INTERFACE ITF_BaseLoggerElement EXTENDS ITF_Base

(*			
	EVERDE sp. z o.o.
	Rafał Osajda		24.03.2025		TC 4024.66
	Definicja nowego zgłoszenia
*)
METHOD PUBLIC EventsDefinition : BOOL
END_METHOD

METHOD PUBLIC GetCode : STRING
VAR_INPUT
END_VAR
END_METHOD

METHOD PUBLIC GetID : UINT
VAR_INPUT
END_VAR
END_METHOD

METHOD PUBLIC GetIdentyfier : ST_BaseElementIdentifier
VAR_INPUT
END_VAR
END_METHOD

METHOD PUBLIC GetName : ST_BaseLabel
VAR_INPUT
END_VAR
END_METHOD

METHOD PUBLIC GetType : E_BaseElementType
VAR_INPUT
END_VAR
END_METHOD

METHOD PUBLIC SetCode
VAR_INPUT
	sCode							: STRING;
	sAdd							: STRING;
END_VAR
END_METHOD

(*			
	EVERDE sp. z o.o.
	Rafał Osajda		03.10.2025		TC 4024.66
	nadawanie unikalnych ID dla zdarzeń
*)
METHOD PUBLIC SetEventsIDs : UINT
VAR_INPUT
	uiNewID		: UINT;
END_VAR
END_METHOD

METHOD PUBLIC SetID : UINT
VAR_INPUT
	uiID					: UINT;
END_VAR
END_METHOD

METHOD PUBLIC SetName
VAR_INPUT
	stName				: ST_BaseLabel;
END_VAR
END_METHOD

METHOD PUBLIC SetType
VAR_INPUT
	eType					: E_BaseElementType;
END_VAR
END_METHOD

END_INTERFACE

(* stored: Version 1.1.0.1
   Itf ITF_BaseLoggerElement: Id {040130d5-be8c-0d8f-3758-2f1440aef3cb}
   Folder ID: Id {ebebc54b-7071-0c25-1f06-3769663c0ef5}
   Method EventsDefinition: Id {9fbb4552-8362-0324-08b0-1fb2884dba78}
   Method GetCode: Id {8b6863d7-2a35-07f8-278a-c5063af13d5f}
   Method GetID: Id {01682019-6db3-0ac2-2322-ec1c5cb9c3b3}
   Method GetIdentyfier: Id {9e739503-7893-0bf4-399c-b179c7bd0bc7}
   Method GetName: Id {878e4ebd-33ce-0ec5-047c-9c76b95779fa}
   Method GetType: Id {c399515a-c57b-0d5c-3183-92e3bee5c2f8}
   Method SetCode: Id {709cb346-bc66-0698-2a3d-3e8bbcb515cf}
   Method SetEventsIDs: Id {7d9014b4-e5ff-0f63-0ed0-28063bd071c8}
   Method SetID: Id {a88625bd-06f5-0c5d-1bbf-fce303221e21}
   Method SetName: Id {29cdd36c-9b48-00dd-03f0-d496e99bfd2c}
   Method SetType: Id {e92df368-a313-0d19-20bc-127474f2c3f1} *)
